// TIA Portal project "babu_3Waytraffic_NewLogic" (V19)

(* hardware
DEVICE "S7-1200 station_1"  S7-1200 Station
   slot 0: "Rack_0"  S7-1200 Rack  Rack  V1.0
   slot 1: "PLC_1"  CPU 1212C DC/DC/DC  6ES7 212-1AE40-0XB0  V4.6
*)

// ===== PLC "PLC_1"  CPU 1212C DC/DC/DC =====

VAR_GLOBAL   // PLC tag table "Default tag table"
   "G3" AT %Q0.0 : Bool;
   "R1" AT %Q0.1 : Bool;
   "R2" AT %Q0.2 : Bool;
   "Y1" AT %Q0.3 : Bool;
   "G1" AT %Q0.4 : Bool;
   "R3" AT %Q0.5 : Bool;
   "Y2" AT %Q0.6 : Bool;
   "G2" AT %Q0.7 : Bool;
   "Y3" AT %Q1.0 : Bool;
   "POWER ON" AT %M0.0 : Bool;
   "MEM" AT %M0.1 : Bool;
   "POWER ON MEM" AT %M0.2 : Bool;
   "G3M" AT %M0.3 : Bool;
   "IP5" AT %M0.4 : Bool;
   "MEM5" AT %M0.5 : Bool;
   "OP5MEM" AT %M0.6 : Bool;
   "IP6" AT %M0.7 : Bool;
   "MEM6" AT %M1.0 : Bool;
   "OP6MEM" AT %M1.1 : Bool;
   "G1M" AT %M1.2 : Bool;
   "G2M" AT %M1.3 : Bool;
   "R1M" AT %M1.4 : Bool;
   "Y1M" AT %M1.5 : Bool;
   "R2M" AT %M1.6 : Bool;
END_VAR

// folder: System blocks/Program resources

DATA_BLOCK "IEC_Timer_0_DB"   // DB1
{ S7_Optimized_Access := 'TRUE' }
AUTHOR : Simatic
FAMILY : IEC
NAME : IEC_TMR
VERSION : 1.0
// stored: InstanceOfName IEC_TIMER
"IEC_TIMER"
BEGIN
END_DATA_BLOCK

DATA_BLOCK "IEC_Timer_0_DB_1"   // DB2
{ S7_Optimized_Access := 'TRUE' }
AUTHOR : Simatic
FAMILY : IEC
NAME : IEC_TMR
VERSION : 1.0
// stored: InstanceOfName IEC_TIMER
"IEC_TIMER"
BEGIN
END_DATA_BLOCK

DATA_BLOCK "IEC_Timer_0_DB_2"   // DB3
{ S7_Optimized_Access := 'TRUE' }
AUTHOR : Simatic
FAMILY : IEC
NAME : IEC_TMR
VERSION : 1.0
// stored: InstanceOfName IEC_TIMER
"IEC_TIMER"
BEGIN
END_DATA_BLOCK

DATA_BLOCK "IEC_Timer_0_DB_3"   // DB4
{ S7_Optimized_Access := 'TRUE' }
AUTHOR : Simatic
FAMILY : IEC
NAME : IEC_TMR
VERSION : 1.0
// stored: InstanceOfName IEC_TIMER
"IEC_TIMER"
BEGIN
END_DATA_BLOCK

DATA_BLOCK "IEC_Timer_0_DB_5"   // DB6
{ S7_Optimized_Access := 'TRUE' }
AUTHOR : Simatic
FAMILY : IEC
NAME : IEC_TMR
VERSION : 1.0
// stored: InstanceOfName IEC_TIMER
"IEC_TIMER"
BEGIN
END_DATA_BLOCK

DATA_BLOCK "IEC_Timer_0_DB_6"   // DB7
{ S7_Optimized_Access := 'TRUE' }
AUTHOR : Simatic
FAMILY : IEC
NAME : IEC_TMR
VERSION : 1.0
// stored: InstanceOfName IEC_TIMER
"IEC_TIMER"
BEGIN
END_DATA_BLOCK

DATA_BLOCK "IEC_Timer_0_DB_7"   // DB8
{ S7_Optimized_Access := 'TRUE' }
AUTHOR : Simatic
FAMILY : IEC
NAME : IEC_TMR
VERSION : 1.0
// stored: InstanceOfName IEC_TIMER
"IEC_TIMER"
BEGIN
END_DATA_BLOCK

DATA_BLOCK "IEC_Timer_0_DB_9"   // DB10
{ S7_Optimized_Access := 'TRUE' }
AUTHOR : Simatic
FAMILY : IEC
NAME : IEC_TMR
VERSION : 1.0
// stored: InstanceOfName IEC_TIMER
"IEC_TIMER"
BEGIN
END_DATA_BLOCK

DATA_BLOCK "IEC_Timer_0_DB_10"   // DB11
{ S7_Optimized_Access := 'TRUE' }
AUTHOR : Simatic
FAMILY : IEC
NAME : IEC_TMR
VERSION : 1.0
// stored: InstanceOfName IEC_TIMER
"IEC_TIMER"
BEGIN
END_DATA_BLOCK

DATA_BLOCK "IEC_Timer_0_DB_11"   // DB12
{ S7_Optimized_Access := 'TRUE' }
AUTHOR : Simatic
FAMILY : IEC
NAME : IEC_TMR
VERSION : 1.0
// stored: InstanceOfName IEC_TIMER
"IEC_TIMER"
BEGIN
END_DATA_BLOCK

DATA_BLOCK "IEC_Timer_0_DB_13"   // DB14
{ S7_Optimized_Access := 'TRUE' }
AUTHOR : Simatic
FAMILY : IEC
NAME : IEC_TMR
VERSION : 1.0
// stored: InstanceOfName IEC_TIMER
"IEC_TIMER"
BEGIN
END_DATA_BLOCK

DATA_BLOCK "IEC_Timer_0_DB_14"   // DB15
{ S7_Optimized_Access := 'TRUE' }
AUTHOR : Simatic
FAMILY : IEC
NAME : IEC_TMR
VERSION : 1.0
// stored: InstanceOfName IEC_TIMER
"IEC_TIMER"
BEGIN
END_DATA_BLOCK

// folder: (top level)

ORGANIZATION_BLOCK "Main"   // OB1, LAD, ProgramCycle
TITLE = "Main Program Sweep (Cycle)"
{ S7_Optimized_Access := 'TRUE' }
VERSION : 0.1
   VAR_INPUT
      Initial_Call : Bool;   // Initial call of this OB
      Remanence : Bool;   // =True, if remanent data are available
   END_VAR
   VAR_TEMP   // added for the SCL form of the ladder/FBD networks
      _w1 : Bool;
   END_VAR
BEGIN

REGION Network 1
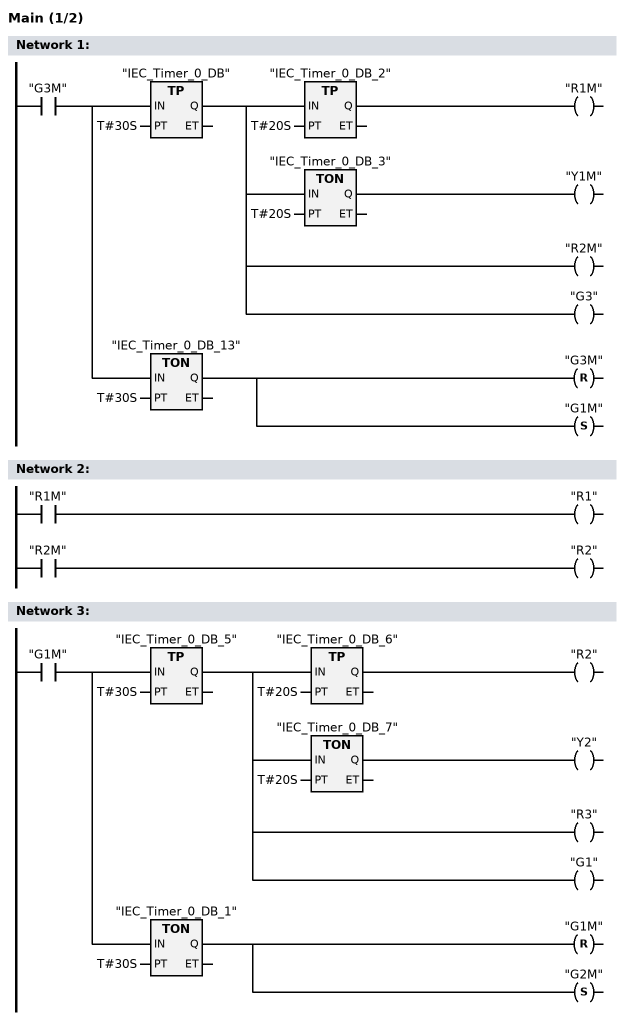
   "IEC_Timer_0_DB".TP(IN := "G3M", PT := T#30S);
   "IEC_Timer_0_DB_2".TP(IN := "IEC_Timer_0_DB".Q, PT := T#20S);
   "R1M" := "IEC_Timer_0_DB_2".Q;
   "IEC_Timer_0_DB_3".TON(IN := "IEC_Timer_0_DB".Q, PT := T#20S);
   "Y1M" := "IEC_Timer_0_DB_3".Q;
   "R2M" := "IEC_Timer_0_DB".Q;
   "G3" := "IEC_Timer_0_DB".Q;
   "IEC_Timer_0_DB_13".TON(IN := "G3M", PT := T#30S);
   IF "IEC_Timer_0_DB_13".Q THEN
       "G3M" := FALSE;
       "G1M" := TRUE;
   END_IF;
END_REGION

REGION Network 2
   RUNG wire#powerrail
      Contact( "R1M" )
      Coil( "R1" )
   END_RUNG
   RUNG wire#powerrail
      Contact( "R2M" )
      Coil( "R2" )
   END_RUNG
   // the same network as SCL:
   "R1" := "R1M";
   "R2" := "R2M";
END_REGION

REGION Network 3
   "IEC_Timer_0_DB_5".TP(IN := "G1M", PT := T#30S);
   "IEC_Timer_0_DB_6".TP(IN := "IEC_Timer_0_DB_5".Q, PT := T#20S);
   "R2" := "IEC_Timer_0_DB_6".Q;
   "IEC_Timer_0_DB_7".TON(IN := "IEC_Timer_0_DB_5".Q, PT := T#20S);
   "Y2" := "IEC_Timer_0_DB_7".Q;
   "R3" := "IEC_Timer_0_DB_5".Q;
   "G1" := "IEC_Timer_0_DB_5".Q;
   "IEC_Timer_0_DB_1".TON(IN := "G1M", PT := T#30S);
   IF "IEC_Timer_0_DB_1".Q THEN
       "G1M" := FALSE;
       "G2M" := TRUE;
   END_IF;
END_REGION

REGION Network 4
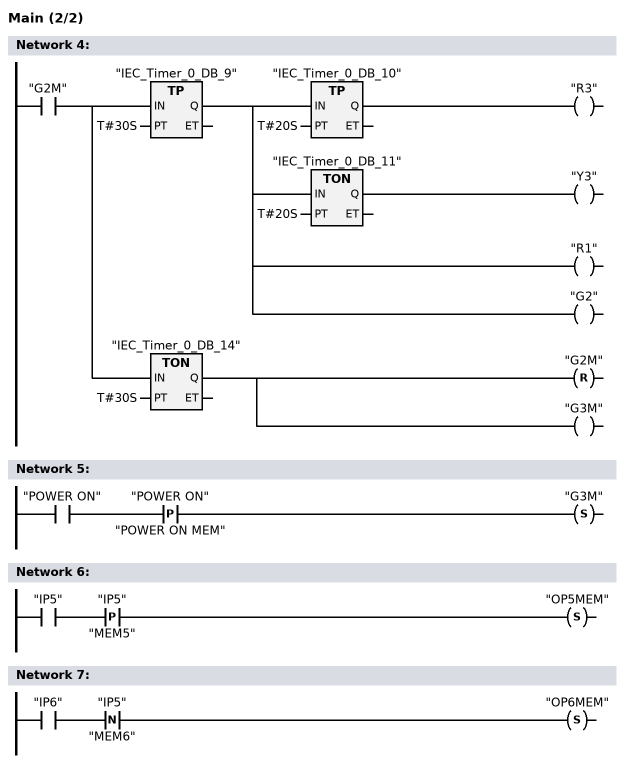
   "IEC_Timer_0_DB_9".TP(IN := "G2M", PT := T#30S);
   "IEC_Timer_0_DB_10".TP(IN := "IEC_Timer_0_DB_9".Q, PT := T#20S);
   "R3" := "IEC_Timer_0_DB_10".Q;
   "IEC_Timer_0_DB_11".TON(IN := "IEC_Timer_0_DB_9".Q, PT := T#20S);
   "Y3" := "IEC_Timer_0_DB_11".Q;
   "R1" := "IEC_Timer_0_DB_9".Q;
   "G2" := "IEC_Timer_0_DB_9".Q;
   "IEC_Timer_0_DB_14".TON(IN := "G2M", PT := T#30S);
   IF "IEC_Timer_0_DB_14".Q THEN "G2M" := FALSE; END_IF;
   "G3M" := "IEC_Timer_0_DB_14".Q;
END_REGION

REGION Network 5
   RUNG wire#powerrail
      Contact( "POWER ON" )
      P_Contact(operand := "POWER ON", bit := "POWER ON MEM")
      S_Coil( "G3M" )
   END_RUNG
   // the same network as SCL:
   #_w1 := "POWER ON" AND "POWER ON" AND NOT "POWER ON MEM";   // rising edge of "POWER ON"
   "POWER ON MEM" := "POWER ON";
   IF #_w1 THEN "G3M" := TRUE; END_IF;
END_REGION

REGION Network 6
   RUNG wire#powerrail
      Contact( "IP5" )
      P_Contact(operand := "IP5", bit := "MEM5")
      S_Coil( "OP5MEM" )
   END_RUNG
   // the same network as SCL:
   #_w1 := "IP5" AND "IP5" AND NOT "MEM5";   // rising edge of "IP5"
   "MEM5" := "IP5";
   IF #_w1 THEN "OP5MEM" := TRUE; END_IF;
END_REGION

REGION Network 7
   RUNG wire#powerrail
      Contact( "IP6" )
      N_Contact(operand := "IP5", bit := "MEM6")
      S_Coil( "OP6MEM" )
   END_RUNG
   // the same network as SCL:
   #_w1 := "IP6" AND NOT "IP5" AND "MEM6";   // falling edge of "IP5"
   "MEM6" := "IP5";
   IF #_w1 THEN "OP6MEM" := TRUE; END_IF;
END_REGION
END_ORGANIZATION_BLOCK